Universal Robots PolyScope program: test.urp

Program test (installation=preprod directory=/programs createdIn=3.14.1.1031110 lastSavedIn=3.14.1.1031110 robotSerialNumber=2020301531)
Calibrated DH parameters: a=[-0.000013, -0.603836, -0.568298, -0.000064, 0.000091, 0]; d=[0.128008, 14.734433, -5.969991, -8.600746, 0.115672, 0.092215]; alpha=[1.570325, -0.007027, -0.006659, 1.569356, -1.5695, 0]; deltaTheta=[-0.000047, -0.169823, 0.067411, 0.102409, -0.00005, 0.00003]
Robot Program (runOnlyOnce=false)
  var_1 := p[-0.2,0.2,0.2,0,3.1415,0]
  MoveJ speed 60 deg/s, acceleration 80 deg/s^2 (useActiveTCP=true)
    Waypoint Waypoint (Variable): variable=var_1
